(* IEC 61131-3 sources: plc-browser-io/CODESYSv3/CODESYS_Control_Win_V3_x64/Application/web_socket, 9 files *)

(* ---- E_WS_Opcode.st ---- *)
{attribute 'qualified_only'}
{attribute 'strict'}
TYPE E_WS_Opcode : (
	CONTINUATION  := 16#00,
	TEXT          := 16#01,
	BINARY        := 16#02,
	CLOSE         := 16#08,
	PING          := 16#09,
	PONG          := 16#0A
)BYTE;
END_TYPE

(* ---- GVL_WebSocket.st ---- *)
{attribute 'qualified_only'}
VAR_GLOBAL
	// ===== WebSocket Server Configuration =====
	uiServerPort       : UINT := 8080;                // TCP listening port
	sServerAddr        : NBS.IP_ADDR := (sAddr := '0.0.0.0'); // Listen on all interfaces

	// ===== Application data (20-byte exchange) =====
	sSendData          : STRING(20) := 'Hello from PLC!     '; // Data to send to browser
	sReceivedData      : STRING(20) := '';                     // Last data received from browser
	xNewDataReceived   : BOOL := FALSE;                        // Flag: new data received
	xSendTrigger       : BOOL := FALSE;                        // Force send sSendData to client

	// ===== Status =====
	xServerRunning     : BOOL := FALSE;
	xClientConnected   : BOOL := FALSE;
	xHandshakeDone     : BOOL := FALSE;
	sLastError         : STRING(80) := '';

	// ===== Debug =====
	uiDebugState       : UINT := 0;
	sDebugInfo         : STRING(255) := '';
END_VAR

(* ---- FC_Base64_Encode.st ---- *)
FUNCTION FC_Base64_Encode : STRING(40)
VAR_INPUT
	pData  : POINTER TO BYTE;  // Pointer to input data
	uiLen  : UINT;             // Length of input data (max ~27 bytes for STRING(40) output)
END_VAR
VAR
	B64    : STRING(64) := 'ABCDEFGHIJKLMNOPQRSTUVWXYZabcdefghijklmnopqrstuvwxyz0123456789+/';
	i      : INT;
	outIdx : INT;
	a      : INT;       // Accumulated bits count
	b      : DWORD;     // Bit buffer
	pSrc   : POINTER TO BYTE;
	val    : INT;
	pOut   : POINTER TO BYTE;
	padCount : INT;
END_VAR

(*
	Synchronous Base64 encoder for raw byte arrays.
	Based on OSCAT BASE64_ENCODE_STREAM logic.
	Used for WebSocket handshake (encoding 20-byte SHA-1 hash -> 28-char base64).
*)

// === IMPLEMENTATION ===
FC_Base64_Encode := '';
pOut := ADR(FC_Base64_Encode);
outIdx := 0;
a := 0;
b := 0;

FOR i := 0 TO UINT_TO_INT(uiLen) - 1 DO
	b := SHL(b, 8) OR BYTE_TO_DWORD(pData[i]);
	a := a + 8;

	WHILE a >= 6 DO
		a := a - 6;
		val := DWORD_TO_INT(SHR(b, a) AND 16#3F);
		// Index into B64 string (1-based in ST)
		pOut[outIdx] := B64[val];
		outIdx := outIdx + 1;
		b := b AND NOT SHL(DWORD#16#FFFFFFFF, a);
	END_WHILE;
END_FOR;

// Handle remaining bits + padding
IF a > 0 THEN
	val := DWORD_TO_INT(SHL(b, 6 - a) AND 16#3F);
	pOut[outIdx] := B64[val];
	outIdx := outIdx + 1;

	// Pad with '=' to make length multiple of 4
	padCount := (4 - (outIdx MOD 4)) MOD 4;
	FOR i := 1 TO padCount DO
		pOut[outIdx] := 61; // '=' = ASCII 61
		outIdx := outIdx + 1;
	END_FOR;
END_IF;

// Null terminator
pOut[outIdx] := 0;

(* ---- FC_SHA1_Bytes.st ---- *)
FUNCTION FC_SHA1_Bytes : BOOL
VAR_INPUT
	pData   : POINTER TO BYTE;  // Pointer to input data
	udiLen  : UDINT;            // Length of input data
END_VAR
VAR_IN_OUT
	abHash  : ARRAY [0..19] OF BYTE;  // Output: 20-byte SHA-1 hash
END_VAR
VAR
	hash    : ARRAY [0..4] OF DWORD;
	w       : ARRAY [0..79] OF DWORD;
	block   : UDINT;
	pos     : UDINT;
	n       : INT;
	n1      : INT;
	a       : DWORD;
	b       : DWORD;
	c       : DWORD;
	d       : DWORD;
	e       : DWORD;
	f       : DWORD;
	k       : DWORD;
	x       : DWORD;
	z       : INT;
	abBuf   : ARRAY [0..63] OF BYTE;
	copyLen : UDINT;
	pSrc    : POINTER TO BYTE;
	pad_done : BOOL;
	totalBlocks : UDINT;
	bytesInLastBlock : UDINT;
	i       : UDINT;
END_VAR

(*
	Synchronous SHA-1 hash computation.
	Based on OSCAT SHA1_STREAM, refactored for single-call usage.
	Used for WebSocket handshake accept key.
*)

// === IMPLEMENTATION ===
// Initialize hash values (SHA-1 constants)
hash[0] := DWORD#16#67452301;
hash[1] := DWORD#16#EFCDAB89;
hash[2] := DWORD#16#98BADCFE;
hash[3] := DWORD#16#10325476;
hash[4] := DWORD#16#C3D2E1F0;

// Calculate number of 64-byte blocks needed
// Message + 1 byte (0x80) + padding + 8 bytes (length)
bytesInLastBlock := (udiLen MOD 64);
IF bytesInLastBlock > 55 THEN
	totalBlocks := (udiLen / 64) + 2;
ELSE
	totalBlocks := (udiLen / 64) + 1;
END_IF;

pos := 0;

FOR block := 0 TO totalBlocks - 1 DO
	// Fill buffer for this block
	FOR n := 0 TO 63 DO
		IF pos + INT_TO_UDINT(n) < udiLen THEN
			// Copy from source data
			abBuf[n] := pData[UDINT_TO_DINT(pos) + n];
		ELSIF pos + INT_TO_UDINT(n) = udiLen AND NOT pad_done THEN
			abBuf[n] := 16#80;
			pad_done := TRUE;
		ELSE
			abBuf[n] := 0;
		END_IF;
	END_FOR;

	// Last block: append bit length in last 8 bytes (big-endian)
	// bitcount = udiLen * 8 = udiLen << 3
	// bytes [56..59] are already 0 (zeroed in loop above)
	// bytes [60..63] encode bits [31..0] of the bit count:
	IF block = totalBlocks - 1 THEN
		abBuf[60] := DWORD_TO_BYTE(SHR(UDINT_TO_DWORD(udiLen), 21)); // bits 31:24 of bitcount
		abBuf[61] := DWORD_TO_BYTE(SHR(UDINT_TO_DWORD(udiLen), 13)); // bits 23:16 of bitcount
		abBuf[62] := DWORD_TO_BYTE(SHR(UDINT_TO_DWORD(udiLen), 5));  // bits 15:8 of bitcount
		abBuf[63] := DWORD_TO_BYTE(SHL(UDINT_TO_DWORD(udiLen), 3));  // bits 7:0 of bitcount
	END_IF;

	pos := pos + 64;

	// Convert byte buffer to 16 DWORDs (big-endian)
	z := 0;
	FOR n1 := 0 TO 15 DO
		w[n1] := SHL(BYTE_TO_DWORD(abBuf[z]), 24)
			OR SHL(BYTE_TO_DWORD(abBuf[z+1]), 16)
			OR SHL(BYTE_TO_DWORD(abBuf[z+2]), 8)
			OR BYTE_TO_DWORD(abBuf[z+3]);
		z := z + 4;
	END_FOR;

	// Extend 16 words to 80 words
	FOR n := 16 TO 79 DO
		w[n] := ROL(w[n-3] XOR w[n-8] XOR w[n-14] XOR w[n-16], 1);
	END_FOR;

	// Initialize working variables
	a := hash[0];
	b := hash[1];
	c := hash[2];
	d := hash[3];
	e := hash[4];

	// Main loop
	FOR n := 0 TO 79 DO
		IF n <= 19 THEN
			f := (b AND c) OR (NOT(b) AND d);
			k := DWORD#16#5A827999;
		ELSIF n <= 39 THEN
			f := b XOR c XOR d;
			k := DWORD#16#6ED9EBA1;
		ELSIF n <= 59 THEN
			f := (b AND c) OR (b AND d) OR (c AND d);
			k := DWORD#16#8F1BBCDC;
		ELSE
			f := b XOR c XOR d;
			k := DWORD#16#CA62C1D6;
		END_IF;

		x := ROL(a, 5) + f + e + k + w[n];
		e := d;
		d := c;
		c := ROL(b, 30);
		b := a;
		a := x;
	END_FOR;

	// Add to hash
	hash[0] := hash[0] + a;
	hash[1] := hash[1] + b;
	hash[2] := hash[2] + c;
	hash[3] := hash[3] + d;
	hash[4] := hash[4] + e;
END_FOR;

// Convert hash DWORDs to byte array (big-endian)
z := 0;
FOR n := 0 TO 4 DO
	FOR n1 := 0 TO 3 DO
		hash[n] := ROL(hash[n], 8);
		abHash[z] := DWORD_TO_BYTE(hash[n]);
		z := z + 1;
	END_FOR;
END_FOR;

FC_SHA1_Bytes := TRUE;

(* ---- FC_WS_BuildAcceptKey.st ---- *)
FUNCTION FC_WS_BuildAcceptKey : STRING(40)
VAR_INPUT
	sClientKey : STRING(40);
	xDebug     : BOOL := TRUE;
END_VAR
VAR
	sGUID       : STRING(40) := '258EAFA5-E914-47DA-95CA-C5AB0DC85B11';
	abHash      : ARRAY [0..19] OF BYTE;
	i           : INT;
	uiKeyLen    : UINT;
	uiGuidLen   : UINT;
	uiTotalLen  : UINT;
	abCombined  : ARRAY [0..79] OF BYTE;
	dwOff       : DWORD;
	pByte       : POINTER TO BYTE;
	pStr        : POINTER TO BYTE;
END_VAR

// === IMPLEMENTATION ===
uiKeyLen  := INT_TO_UINT(LEN(sClientKey));
uiGuidLen := INT_TO_UINT(LEN(sGUID));
uiTotalLen := uiKeyLen + uiGuidLen;

// Log input key details
IF xDebug THEN
	LogComponent.Logger.LogADD(Component:= LogComponent.WS, LogClass:= cmplog.LogClass.LOG_INFO,
		Message:= CONCAT('BuildAcceptKey: keyLen=', TO_STRING(uiKeyLen)));
	LogComponent.Logger.LogADD(Component:= LogComponent.WS, LogClass:= cmplog.LogClass.LOG_INFO,
		Message:= CONCAT('BuildAcceptKey: key=[', CONCAT(sClientKey, ']')));
	LogComponent.Logger.LogADD(Component:= LogComponent.WS, LogClass:= cmplog.LogClass.LOG_INFO,
		Message:= CONCAT('BuildAcceptKey: totalLen=', TO_STRING(uiTotalLen)));
END_IF;

// Copy client key bytes into combined buffer
pStr := ADR(sClientKey);
FOR i := 0 TO UINT_TO_INT(uiKeyLen) - 1 DO
	dwOff := INT_TO_DWORD(i);
	pByte := pStr + dwOff;
	abCombined[i] := pByte^;
END_FOR;

// Copy GUID bytes after the key
pStr := ADR(sGUID);
FOR i := 0 TO UINT_TO_INT(uiGuidLen) - 1 DO
	dwOff := INT_TO_DWORD(i);
	pByte := pStr + dwOff;
	abCombined[UINT_TO_INT(uiKeyLen) + i] := pByte^;
END_FOR;

// SHA-1 hash
FC_SHA1_Bytes(
	pData  := ADR(abCombined),
	udiLen := UINT_TO_UDINT(uiTotalLen),
	abHash := abHash
);

// Log first 4 bytes of SHA1 as hex for verification
IF xDebug THEN
	LogComponent.Logger.LogADD(Component:= LogComponent.WS, LogClass:= cmplog.LogClass.LOG_INFO,
		Message:= CONCAT('SHA1[0..3]: ',
			CONCAT(TO_STRING(abHash[0]), CONCAT(' ',
			CONCAT(TO_STRING(abHash[1]), CONCAT(' ',
			CONCAT(TO_STRING(abHash[2]), CONCAT(' ',
			TO_STRING(abHash[3])))))))));
END_IF;

// Base64 encode 20-byte hash
FC_WS_BuildAcceptKey := FC_Base64_Encode(
	pData := ADR(abHash),
	uiLen := 20
);

LogComponent.Logger.LogADD(Component:= LogComponent.WS, LogClass:= cmplog.LogClass.LOG_INFO,
	Message:= CONCAT('BuildAcceptKey result: ', FC_WS_BuildAcceptKey));

(* ---- FC_WS_BuildFrame.st ---- *)
FUNCTION FC_WS_BuildFrame : UINT
VAR_INPUT
	eOpcode     : E_WS_Opcode;         // Frame opcode
	pPayload    : POINTER TO BYTE;     // Pointer to payload data
	uiPayloadLen: UINT;                // Payload length
	xFin        : BOOL := TRUE;        // FIN bit (TRUE = final frame)
END_VAR
VAR_IN_OUT
	abOutBuf    : ARRAY [0..1023] OF BYTE;  // Output: built frame
END_VAR
VAR
	idx       : UINT;
	i         : UINT;
	byte0     : BYTE;
	pSrc      : POINTER TO BYTE;
END_VAR

(*
	Builds a WebSocket frame for SENDING from server to client.
	Server frames are NOT masked (RFC 6455 Section 5.1).
	Returns total frame length in bytes.
*)

// === IMPLEMENTATION ===
idx := 0;

// Byte 0: FIN + Opcode
byte0 := eOpcode;
IF xFin THEN
	byte0 := byte0 OR 16#80;
END_IF;
abOutBuf[0] := byte0;
idx := 1;

// Byte 1+: Payload length (no mask bit for server frames)
IF uiPayloadLen < 126 THEN
	abOutBuf[1] := UINT_TO_BYTE(uiPayloadLen);
	idx := 2;
ELSIF uiPayloadLen < 65535 THEN
	abOutBuf[1] := 126;
	abOutBuf[2] := UINT_TO_BYTE(SHR(uiPayloadLen, 8));
	abOutBuf[3] := UINT_TO_BYTE(uiPayloadLen AND 16#FF);
	idx := 4;
END_IF;

// Copy payload data
FOR i := 0 TO uiPayloadLen - 1 DO
	IF UINT_TO_INT(idx + i) > 1023 THEN
		EXIT;
	END_IF;
	abOutBuf[idx + i] := pPayload[i];
END_FOR;

FC_WS_BuildFrame := idx + uiPayloadLen;

(* ---- FC_WS_ParseFrame.st ---- *)
FUNCTION FC_WS_ParseFrame : BOOL
VAR_INPUT
	pData     : POINTER TO BYTE;
	uiDataLen : UINT;
END_VAR
VAR_IN_OUT
	stFrame   : ST_WS_Frame;
END_VAR
VAR
	byte0       : BYTE;
	byte1       : BYTE;
	payloadLen7 : BYTE;
	maskStart   : UINT;
	payloadStart: UINT;
	i           : UINT;
	dwOff       : DWORD;
	pByte       : POINTER TO BYTE;
	bMaskIdx    : INT;
END_VAR

// === IMPLEMENTATION ===
FC_WS_ParseFrame := FALSE;
stFrame.xValid := FALSE;

IF uiDataLen < 2 THEN
	RETURN;
END_IF;

// Read byte 0 and byte 1 using direct pointer offset
byte0 := pData^;
dwOff := 1;
pByte := pData + dwOff;
byte1 := pByte^;

// Parse header fields
stFrame.xFin    := (byte0 AND 16#80) = 16#80;
stFrame.xMasked := (byte1 AND 16#80) = 16#80;

// Opcode - cast via BYTE to avoid strict enum error
CASE BYTE_TO_INT(byte0 AND 16#0F) OF
	0:  stFrame.eOpcode := E_WS_Opcode.CONTINUATION;
	1:  stFrame.eOpcode := E_WS_Opcode.TEXT;
	2:  stFrame.eOpcode := E_WS_Opcode.BINARY;
	8:  stFrame.eOpcode := E_WS_Opcode.CLOSE;
	9:  stFrame.eOpcode := E_WS_Opcode.PING;
	10: stFrame.eOpcode := E_WS_Opcode.PONG;
ELSE
	stFrame.eOpcode := E_WS_Opcode.CONTINUATION;
END_CASE;

payloadLen7 := byte1 AND 16#7F;

IF payloadLen7 < 126 THEN
	stFrame.udiPayloadLen := BYTE_TO_UDINT(payloadLen7);
	maskStart := 2;
ELSIF payloadLen7 = 126 THEN
	IF uiDataLen < 4 THEN RETURN; END_IF;
	dwOff := 2; pByte := pData + dwOff;
	stFrame.udiPayloadLen := SHL(BYTE_TO_UDINT(pByte^), 8);
	dwOff := 3; pByte := pData + dwOff;
	stFrame.udiPayloadLen := stFrame.udiPayloadLen OR BYTE_TO_UDINT(pByte^);
	maskStart := 4;
ELSE
	IF uiDataLen < 10 THEN RETURN; END_IF;
	dwOff := 6; pByte := pData + dwOff; stFrame.udiPayloadLen := SHL(BYTE_TO_UDINT(pByte^), 24);
	dwOff := 7; pByte := pData + dwOff; stFrame.udiPayloadLen := stFrame.udiPayloadLen OR SHL(BYTE_TO_UDINT(pByte^), 16);
	dwOff := 8; pByte := pData + dwOff; stFrame.udiPayloadLen := stFrame.udiPayloadLen OR SHL(BYTE_TO_UDINT(pByte^), 8);
	dwOff := 9; pByte := pData + dwOff; stFrame.udiPayloadLen := stFrame.udiPayloadLen OR BYTE_TO_UDINT(pByte^);
	maskStart := 10;
END_IF;

IF stFrame.xMasked THEN
	IF uiDataLen < maskStart + 4 THEN RETURN; END_IF;
	dwOff := UINT_TO_DWORD(maskStart);     pByte := pData + dwOff; stFrame.abMaskKey[0] := pByte^;
	dwOff := UINT_TO_DWORD(maskStart + 1); pByte := pData + dwOff; stFrame.abMaskKey[1] := pByte^;
	dwOff := UINT_TO_DWORD(maskStart + 2); pByte := pData + dwOff; stFrame.abMaskKey[2] := pByte^;
	dwOff := UINT_TO_DWORD(maskStart + 3); pByte := pData + dwOff; stFrame.abMaskKey[3] := pByte^;
	payloadStart := maskStart + 4;
ELSE
	stFrame.abMaskKey[0] := 0;
	stFrame.abMaskKey[1] := 0;
	stFrame.abMaskKey[2] := 0;
	stFrame.abMaskKey[3] := 0;
	payloadStart := maskStart;
END_IF;

// Validate length
stFrame.uiTotalLen := payloadStart + UDINT_TO_UINT(stFrame.udiPayloadLen);
IF UINT_TO_UDINT(uiDataLen) < UINT_TO_UDINT(payloadStart) + stFrame.udiPayloadLen THEN
	RETURN;
END_IF;
IF stFrame.udiPayloadLen > 1024 THEN
	stFrame.udiPayloadLen := 1024;
END_IF;

// Read and unmask payload (skip if payload is empty, e.g. CLOSE/PING)
IF stFrame.udiPayloadLen > 0 THEN
	FOR i := 0 TO UDINT_TO_UINT(stFrame.udiPayloadLen) - 1 DO
		dwOff := UINT_TO_DWORD(payloadStart + i);
		pByte := pData + dwOff;
		bMaskIdx := UINT_TO_INT(i MOD 4);
		IF stFrame.xMasked THEN
			stFrame.abPayload[i] := pByte^ XOR stFrame.abMaskKey[bMaskIdx];
		ELSE
			stFrame.abPayload[i] := pByte^;
		END_IF;
	END_FOR;
END_IF;

stFrame.xValid := TRUE;
FC_WS_ParseFrame := TRUE;

(* ---- FB_WebSocket_Server.st ---- *)
FUNCTION_BLOCK FB_WebSocket_Server
VAR_INPUT
	xEnable      : BOOL;
	ipAddr       : NBS.IP_ADDR;
	uiPort       : UINT := 8080;
	pSendData    : POINTER TO BYTE;
	uiSendSize   : UINT := 0;
	xSendTrigger : BOOL;

	pRecvData    : POINTER TO BYTE;
	uiRecvSize   : UINT := 0;
	xDebug       : BOOL := TRUE;
END_VAR

VAR_OUTPUT
	xRunning         : BOOL;
	xClientConnected : BOOL;
	xHandshakeOK     : BOOL;
	uiReceivedLen    : UINT;
	xNewDataReceived : BOOL;
	eState           : E_WS_State;
	sError           : STRING(80);
END_VAR

VAR
	fbServer     : NBS.TCP_Server;
	fbConnection : NBS.TCP_Connection;
	fbRead       : NBS.TCP_Read;
	fbWrite      : NBS.TCP_Write;

	eStep          : E_WS_State := E_WS_State.IDLE;
	eStepAfterSend : E_WS_State;

	abRecvBuf    : ARRAY [0..2047] OF BYTE;
	abSendBuf    : ARRAY [0..2047] OF BYTE;
	uiRecvLen    : UINT;
	uiSendLen    : UINT;

	stFrame      : ST_WS_Frame;
	abFrameBuf   : ARRAY [0..1023] OF BYTE;
	uiFrameLen   : UINT;

	sClientKey   : STRING(40);
	sAcceptKey   : STRING(40);
	sResponse    : STRING(255);
	uiResponseLen: UINT;

	abPayloadOut : ARRAY [0..31] OF BYTE;

	i     : INT;
	dwOff : DWORD;
	pByte : POINTER TO BYTE;
	pStr  : POINTER TO BYTE;

	xSendTrigLast : BOOL;
	xEnableLast   : BOOL;
	xSendPending  : BOOL;
	sLogMsg       : STRING(255);
END_VAR

// === IMPLEMENTATION ===
// ALWAYS call maintenance blocks if server is starting or running
IF eStep <> E_WS_State.IDLE THEN
	fbServer(xEnable := TRUE, ipAddr := ipAddr, uiPort := uiPort);
	fbConnection(xEnable := TRUE, hServer := fbServer.hServer);
END_IF;

// Trigger detection
IF xSendTrigger AND NOT xSendTrigLast THEN
	xSendPending := TRUE;
END_IF;
xSendTrigLast := xSendTrigger;

// Global disable
IF NOT xEnable AND eStep <> E_WS_State.IDLE AND eStep <> E_WS_State.CLOSING THEN
	sError := 'User disabled server';
	eStep := E_WS_State.WS_SEND_CLOSE;
END_IF;

xNewDataReceived := FALSE;

CASE eStep OF
// ... (IDLE, SERVER_STARTING etc)
E_WS_State.IDLE:
	xRunning := FALSE;
	xClientConnected := FALSE;
	xHandshakeOK := FALSE;
	sError := '';
	IF xEnable THEN
		eStep := E_WS_State.SERVER_STARTING;
	END_IF;
// ...
E_WS_State.SERVER_STARTING:
	IF fbServer.xError THEN
		sError := 'TCP_Server failed';
		eStep := E_WS_State.ERROR;
	ELSIF fbServer.hServer <> 0 THEN
		xRunning := TRUE;
		eStep := E_WS_State.CONN_WAITING;
	END_IF;
// ...
E_WS_State.CONN_WAITING:
	IF fbConnection.xActive THEN
		xClientConnected := TRUE;
		eStep := E_WS_State.HANDSHAKE_READ;
	ELSIF fbConnection.xError THEN
		sError := 'TCP_Connection error';
		eStep := E_WS_State.ERROR;
	END_IF;

// --------------------------------------------------
E_WS_State.HANDSHAKE_READ:
	fbRead(
		xEnable     := TRUE,
		hConnection := fbConnection.hConnection,
		szSize      := SIZEOF(abRecvBuf),
		pData       := ADR(abRecvBuf)
	);
	IF fbRead.xReady AND fbRead.szCount > 0 THEN
		uiRecvLen := TO_UINT(fbRead.szCount);
		fbRead(xEnable := FALSE);
		eStep := E_WS_State.HANDSHAKE_PARSE;
	ELSIF fbRead.xError THEN
		sError := 'Handshake read error';
		eStep := E_WS_State.CLOSING;
	END_IF;

// --------------------------------------------------
E_WS_State.HANDSHAKE_PARSE:
	sClientKey := FC_ExtractWSKey(pData := ADR(abRecvBuf), uiDataLen := uiRecvLen);
	IF LEN(sClientKey) = 0 THEN
		sError := 'No WS key found';
		eStep := E_WS_State.CLOSING;
	ELSE
		sAcceptKey := FC_WS_BuildAcceptKey(sClientKey := sClientKey, xDebug := xDebug);
		sResponse := 'HTTP/1.1 101 Switching Protocols$0D$0A';
		sResponse := CONCAT(sResponse, 'Upgrade: websocket$0D$0A');
		sResponse := CONCAT(sResponse, 'Connection: Upgrade$0D$0A');
		sResponse := CONCAT(sResponse, 'Sec-WebSocket-Accept: ');
		sResponse := CONCAT(sResponse, sAcceptKey);
		sResponse := CONCAT(sResponse, '$0D$0A$0D$0A');

		uiResponseLen := INT_TO_UINT(LEN(sResponse));
		pStr := ADR(sResponse);
		FOR i := 0 TO UINT_TO_INT(uiResponseLen) - 1 DO
			abSendBuf[i] := pStr[i];
		END_FOR;
		uiSendLen := uiResponseLen;
		eStep := E_WS_State.HANDSHAKE_SEND;
	END_IF;

// --------------------------------------------------
E_WS_State.HANDSHAKE_SEND:
	fbWrite(
		xExecute    := TRUE,
		hConnection := fbConnection.hConnection,
		szSize      := TO_UDINT(uiSendLen),
		pData       := ADR(abSendBuf)
	);
	IF fbWrite.xDone THEN
		fbWrite(xExecute := FALSE);
		eStep := E_WS_State.WS_CONNECTED;
	ELSIF fbWrite.xError THEN
		sError := 'Handshake send failed';
		eStep := E_WS_State.CLOSING;
	END_IF;

// --------------------------------------------------
E_WS_State.WS_CONNECTED:
	xHandshakeOK := TRUE;
	IF NOT fbConnection.xActive THEN
		sError := 'Connection lost';
		eStep := E_WS_State.CLOSING;
	END_IF;

// --------------------------------------------------
E_WS_State.WS_SEND_CLOSE:
	// Build Close frame (opcode 0x8)
	uiFrameLen := FC_WS_BuildFrame(
		eOpcode := E_WS_Opcode.CLOSE,
		pPayload := ADR(abFrameBuf), // empty payload
		uiPayloadLen := 0,
		xFin := TRUE,
		abOutBuf := abFrameBuf
	);

	FOR i := 0 TO UINT_TO_INT(uiFrameLen) - 1 DO
		abSendBuf[i] := abFrameBuf[i];
	END_FOR;
	uiSendLen := uiFrameLen;

	LogComponent.Logger.LogADD(Component:= LogComponent.WS, LogClass:= cmplog.LogClass.LOG_INFO,
		Message:= 'WS Send: Close frame');

	fbWrite(
		xExecute := TRUE,
		hConnection := fbConnection.hConnection,
		szSize := TO_UDINT(uiSendLen),
		pData := ADR(abSendBuf)
	);

	IF fbWrite.xDone THEN
		fbWrite(xExecute := FALSE);
		eStep := E_WS_State.CLOSING;
	ELSIF fbWrite.xError THEN
		fbWrite(xExecute := FALSE);
		eStep := E_WS_State.CLOSING; // Close anyway on error
	END_IF;

// --------------------------------------------------
E_WS_State.CLOSING:
	fbRead(xEnable := FALSE);
	fbWrite(xExecute := FALSE);
	fbConnection(xEnable := FALSE);
	fbServer(xEnable := FALSE);
	eStep := E_WS_State.IDLE;

// --------------------------------------------------
E_WS_State.ERROR:
	xRunning := FALSE;
	IF NOT xEnable THEN
		eStep := E_WS_State.IDLE;
	END_IF;

END_CASE;

// ==================================================
// FULL-DUPLEX DATA EXCHANGE (Runs when connected)
// ==================================================
IF eStep = E_WS_State.WS_CONNECTED THEN

	// --- 1. RECEIVER ---
	fbRead(
		xEnable := TRUE,
		hConnection := fbConnection.hConnection,
		szSize := SIZEOF(abRecvBuf),
		pData := ADR(abRecvBuf)
	);

	IF fbRead.xReady AND fbRead.szCount > 0 THEN
		uiRecvLen := TO_UINT(fbRead.szCount);

		IF xDebug THEN
			// Log raw bytes for debugging
			sLogMsg := CONCAT('RX raw: len=', TO_STRING(uiRecvLen));
			sLogMsg := CONCAT(sLogMsg, CONCAT(' b0=', TO_STRING(abRecvBuf[0])));
			sLogMsg := CONCAT(sLogMsg, CONCAT(' b1=', TO_STRING(abRecvBuf[1])));
			LogComponent.Logger.LogADD(Component:= LogComponent.WS, LogClass:= cmplog.LogClass.LOG_INFO, Message:= sLogMsg);
		END_IF;

		IF FC_WS_ParseFrame(pData := ADR(abRecvBuf), uiDataLen := uiRecvLen, stFrame := stFrame) THEN
			IF xDebug THEN
				sLogMsg := CONCAT('Parsed opcode=', TO_STRING(stFrame.eOpcode));
				sLogMsg := CONCAT(sLogMsg, CONCAT(' payloadLen=', TO_STRING(stFrame.udiPayloadLen)));
				LogComponent.Logger.LogADD(Component:= LogComponent.WS, LogClass:= cmplog.LogClass.LOG_INFO, Message:= sLogMsg);
			END_IF;

			CASE stFrame.eOpcode OF
				E_WS_Opcode.TEXT, E_WS_Opcode.BINARY:
					IF pRecvData <> 0 AND uiRecvSize > 0 THEN
						uiReceivedLen := MIN(UDINT_TO_UINT(stFrame.udiPayloadLen), uiRecvSize);
						FOR i := 0 TO UINT_TO_INT(uiReceivedLen) - 1 DO
							pRecvData[i] := stFrame.abPayload[i];
						END_FOR;
						xNewDataReceived := TRUE;
					END_IF;

					IF xDebug THEN
						LogComponent.Logger.LogADD(Component:= LogComponent.WS, LogClass:= cmplog.LogClass.LOG_INFO,
							Message:= CONCAT('WS Recv: Binary Map Size=', TO_STRING(uiReceivedLen)));
					END_IF;

				E_WS_Opcode.CLOSE:
					IF xDebug THEN
						LogComponent.Logger.LogADD(Component:= LogComponent.WS, LogClass:= cmplog.LogClass.LOG_WARNING,
							Message:= 'Got CLOSE frame from client');
					END_IF;
					sError := 'Client requested close';
					fbRead(xEnable := FALSE);
					eStep := E_WS_State.WS_SEND_CLOSE;

				E_WS_Opcode.PING:
					IF xDebug THEN
						LogComponent.Logger.LogADD(Component:= LogComponent.WS, LogClass:= cmplog.LogClass.LOG_INFO,
							Message:= 'Got PING frame');
					END_IF;
			END_CASE;
		ELSE
			IF xDebug THEN
				LogComponent.Logger.LogADD(Component:= LogComponent.WS, LogClass:= cmplog.LogClass.LOG_WARNING,
					Message:= CONCAT('ParseFrame FAILED, len=', TO_STRING(uiRecvLen)));
			END_IF;
		END_IF;
	ELSIF fbRead.xError THEN
		IF xDebug THEN
			sLogMsg := CONCAT('fbRead ERROR eError=', TO_STRING(fbRead.eError));
			LogComponent.Logger.LogADD(Component:= LogComponent.WS, LogClass:= cmplog.LogClass.LOG_ERROR, Message:= sLogMsg);
		END_IF;
		sError := 'Read error';
		eStep := E_WS_State.CLOSING;
	END_IF;

	// --- 2. TRANSMITTER ---
	IF xSendPending AND NOT fbWrite.xBusy THEN
		IF pSendData <> 0 AND uiSendSize > 0 THEN
			uiFrameLen := FC_WS_BuildFrame(
				eOpcode := E_WS_Opcode.BINARY,
				pPayload := pSendData,
				uiPayloadLen := uiSendSize,
				xFin := TRUE,
				abOutBuf := abFrameBuf
			);

			FOR i := 0 TO UINT_TO_INT(uiFrameLen) - 1 DO
				abSendBuf[i] := abFrameBuf[i];
			END_FOR;
			uiSendLen := uiFrameLen;

			fbWrite(xExecute := TRUE, hConnection := fbConnection.hConnection, szSize := TO_UDINT(uiSendLen), pData := ADR(abSendBuf));
			xSendPending := FALSE;

			IF xDebug THEN
				LogComponent.Logger.LogADD(Component:= LogComponent.WS, LogClass:= cmplog.LogClass.LOG_INFO,
					Message:= CONCAT('WS Send: Binary Size=', TO_STRING(uiSendSize)));
			END_IF;
		ELSE
			xSendPending := FALSE; // Nothing to send
		END_IF;

	ELSIF fbWrite.xDone OR fbWrite.xError THEN
		fbWrite(xExecute := FALSE);
	ELSE
		fbWrite();
	END_IF;

END_IF;

eState := eStep;
// Update GVL info
GVL_WebSocket.sDebugInfo := CONCAT('Step: ', TO_STRING(eStep));
GVL_WebSocket.sDebugInfo := CONCAT(GVL_WebSocket.sDebugInfo, ' | Cnt: ');
GVL_WebSocket.sDebugInfo := CONCAT(GVL_WebSocket.sDebugInfo, TO_STRING(fbConnection.xActive));

(* ---- Web_socket_programm_call.st ---- *)
PROGRAM Web_socket_programm_call
VAR
	fbWS          : FB_WebSocket_Server;
	xStart        : BOOL := TRUE;          // Set TRUE to start server

	stSimInputs   : ST_SimulationInputs;  // Data FROM Browser
	stSimOutputs  : ST_SimulationOutputs; // Data TO Browser

	// Watchdog logic
	uiLastWD      : BYTE;
	tonWD         : TON;
	xCommError    : BOOL;

	// Cyclic transmission
	tonSend       : TON;
END_VAR

// === IMPLEMENTATION ===

// 1. Increment Watchdog for Browser
stSimOutputs.uiWatchdog_Outputs := stSimOutputs.uiWatchdog_Outputs + 1;

// 2. Monitoring Watchdog from Browser
IF stSimInputs.uiWatchdog_Inputs <> uiLastWD THEN
	uiLastWD := stSimInputs.uiWatchdog_Inputs;
	tonWD(IN := FALSE); // Reset timer
END_IF;

tonWD(IN := TRUE, PT := T#1000MS); // Default 1s, can be changed based on JSON
xCommError := tonWD.Q;

// 3. Cyclic Send (target 10ms)
tonSend(IN := NOT tonSend.Q, PT := T#10MS);

// 4. WebSocket Server Call
fbWS(
	xEnable      := xStart,
	ipAddr       := GVL_WebSocket.sServerAddr,
	uiPort       := GVL_WebSocket.uiServerPort,
	pSendData    := ADR(stSimOutputs),
	uiSendSize   := SIZEOF(stSimOutputs),
	xSendTrigger := tonSend.Q,
	pRecvData    := ADR(stSimInputs),
	uiRecvSize   := SIZEOF(stSimInputs)
);

// 5. Global Status Update
GVL_WebSocket.xServerRunning   := fbWS.xRunning;
GVL_WebSocket.xClientConnected := fbWS.xClientConnected;
GVL_WebSocket.xHandshakeDone   := fbWS.xHandshakeOK;
GVL_WebSocket.uiDebugState     := fbWS.eState;
GVL_WebSocket.sLastError       := fbWS.sError;

IF fbWS.xNewDataReceived THEN
	GVL_WebSocket.xNewDataReceived  := TRUE;
	// Log for confirmation (optional, might be heavy at 10ms)
	// LogComponent.Logger.LogADD(Component:= LogComponent.WS, LogClass:= cmplog.LogClass.LOG_INFO, Message:= 'Data Sync OK');
ELSE
	GVL_WebSocket.xNewDataReceived := FALSE;
END_IF;
